{attribute 'qualified_only'}
{attribute 'strict'}
TYPE E_SCANNER_Baudrate :
(
	IDLE,
	READ,
	WRITE,
	READERROR,
	WRITEERROR,
	DONE
);
END_TYPE

(* stored: Version 1.1.0.1
   DUT E_SCANNER_Baudrate: Id {feddf96c-9938-4580-a3fc-ff1040328cdd} *)
